# EPICS autosave request: energy_meter/autoSaveRestore/energy_meter.req
$(device):CalibrationFactor
